INTERFACE PUBLIC I_AsyncCommandStateControl

METHOD PUBLIC Error
VAR_INPUT
	errorId : UDINT;
END_VAR
END_METHOD

METHOD PUBLIC Next
END_METHOD

END_INTERFACE

(* stored: Version 1.1.0.1, ProductVersion 3.1.4024.12
   Itf I_AsyncCommandStateControl: Id {e47154c6-4a1f-07f5-0779-c72fb0d71966}
   Method Error: Id {4be21d91-50c2-0277-0428-d7da6a12265f}
   Method Next: Id {5d7fa840-69e3-03ca-3870-3879c65f0611} *)
